SUBAPPLICATION Ventilsteuerung_Uebung_020e (* DigitalInput_I1 auf DigitalOutput_Q1; E_TOF; Ausschaltverzögert *)
  (* Standard: 61499-2 *)
  (* Version 1.0, 2023-10-23, franz *)
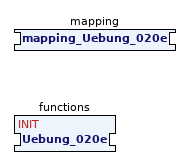
  SUBAPPS
    mapping : mapping_Uebung_020e;
    functions : Uebung_020e;
  END_SUBAPPS
END_SUBAPPLICATION
